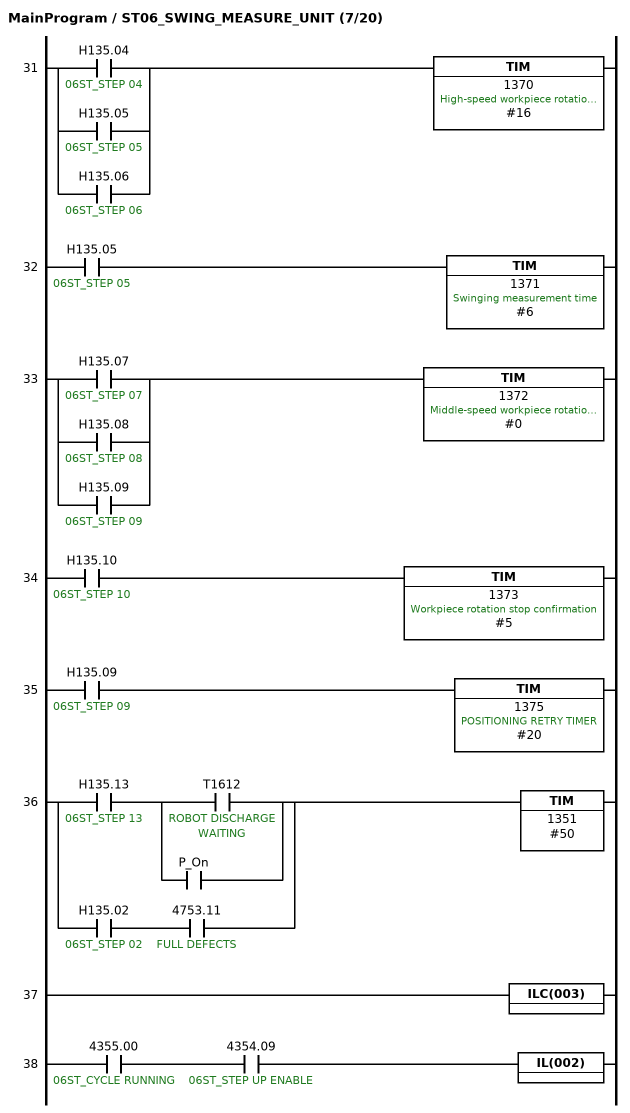
; [picture p360: MainProgram / ST06_SWING_MEASURE_UNIT, rungs 31-38]
; rung 31
LD H135.04  ; 06ST_STEP 04
OR H135.05  ; 06ST_STEP 05
OR H135.06  ; 06ST_STEP 06
TIM 1370 #16  ; High-speed workpiece rotation stability  // #15 => #8
; rung 32
LD H135.05  ; 06ST_STEP 05
TIM 1371 #6  ; Swinging measurement time
; rung 33
LD H135.07  ; 06ST_STEP 07
OR H135.08  ; 06ST_STEP 08
OR H135.09  ; 06ST_STEP 09
TIM 1372 #0  ; Middle-speed workpiece rotation stability
; rung 34
LD H135.10  ; 06ST_STEP 10
TIM 1373 #5  ; Workpiece rotation stop confirmation
; rung 35
LD H135.09  ; 06ST_STEP 09
TIM 1375 #20  ; POSITIONING RETRY TIMER
; rung 36
LD H135.13  ; 06ST_STEP 13
LD T1612  ; ROBOT DISCHARGE WAITING
OR P_On
ANDLD
LD H135.02  ; 06ST_STEP 02
AND 4753.11  ; FULL DEFECTS
ORLD
TIM 1351 #50
; rung 37
ILC(003)
; rung 38
LD 4355.00  ; 06ST_CYCLE RUNNING
AND 4354.09  ; 06ST_STEP UP ENABLE
IL(002)

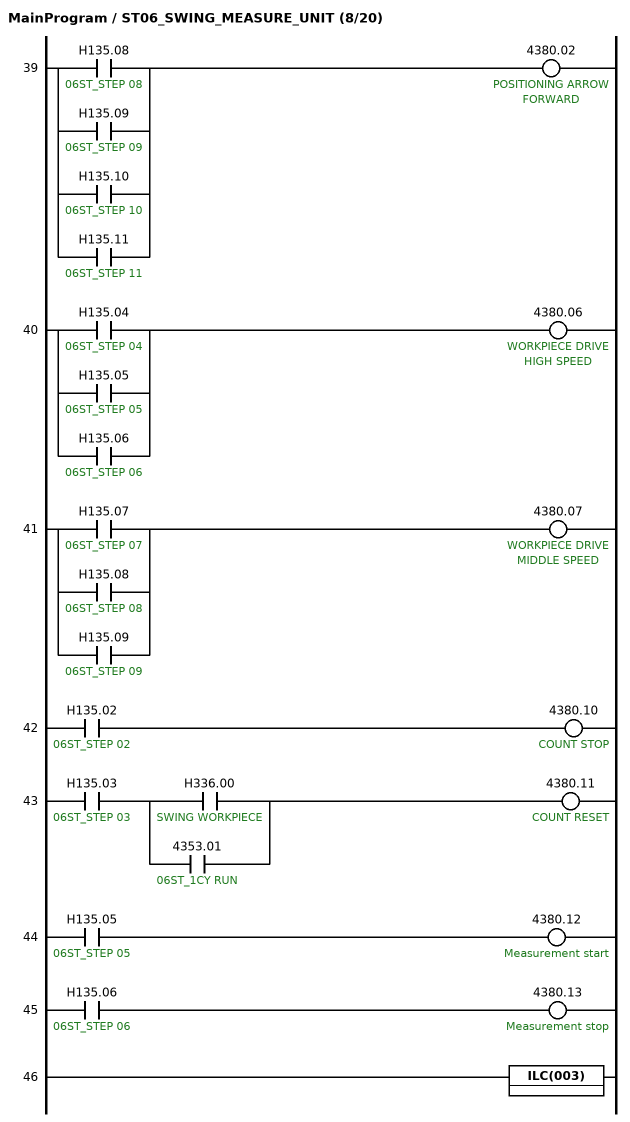
; rung 39
LD H135.08  ; 06ST_STEP 08
OR H135.09  ; 06ST_STEP 09
OR H135.10  ; 06ST_STEP 10
OR H135.11  ; 06ST_STEP 11
OUT 4380.02  ; POSITIONING ARROW FORWARD
; rung 40
LD H135.04  ; 06ST_STEP 04
OR H135.05  ; 06ST_STEP 05
OR H135.06  ; 06ST_STEP 06
OUT 4380.06  ; WORKPIECE DRIVE HIGH SPEED
; rung 41
LD H135.07  ; 06ST_STEP 07
OR H135.08  ; 06ST_STEP 08
OR H135.09  ; 06ST_STEP 09
OUT 4380.07  ; WORKPIECE DRIVE MIDDLE SPEED
; rung 42
LD H135.02  ; 06ST_STEP 02
OUT 4380.10  ; COUNT STOP
; rung 43
LD H135.03  ; 06ST_STEP 03
LD H336.00  ; SWING WORKPIECE
OR 4353.01  ; 06ST_1CY RUN
ANDLD
OUT 4380.11  ; COUNT RESET
; rung 44
LD H135.05  ; 06ST_STEP 05
OUT 4380.12  ; Measurement start
; rung 45
LD H135.06  ; 06ST_STEP 06
OUT 4380.13  ; Measurement stop
; rung 46
ILC(003)

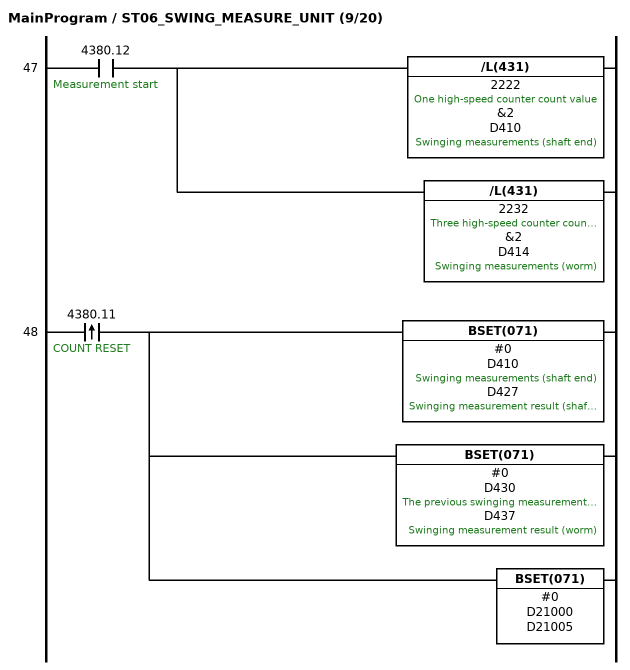
; rung 47
LD 4380.12  ; Measurement start
/L(431) 2222 &2 D410  ; One high-speed counter count value, Swinging measurements (shaft end)
/L(431) 2232 &2 D414  ; Three high-speed counter count value, Swinging measurements (worm)
; rung 48
@LD 4380.11  ; COUNT RESET
BSET(071) #0 D410 D427  ; Swinging measurements (shaft end), Swinging measurement result (shaft end)
BSET(071) #0 D430 D437  ; The previous swinging measurements (worm), Swinging measurement result (worm)
BSET(071) #0 D21000 D21005

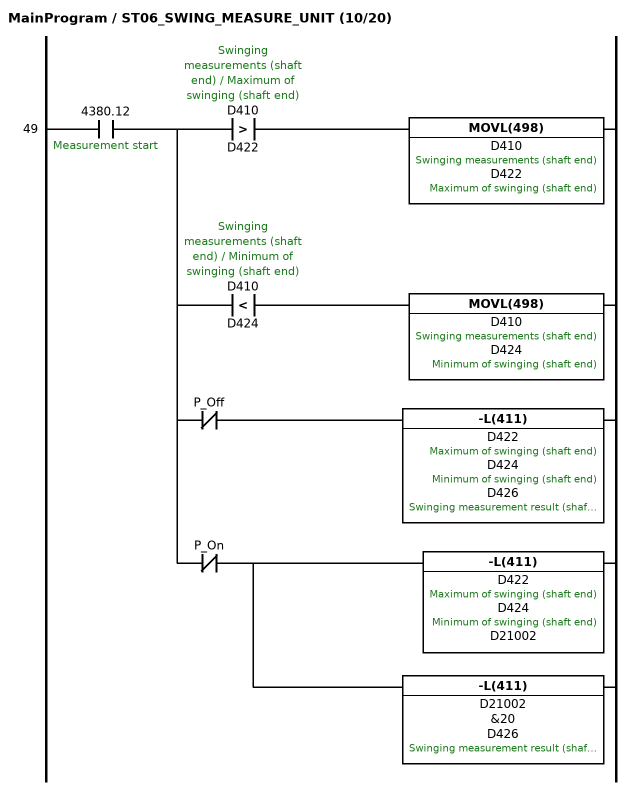
; rung 49
LD 4380.12  ; Measurement start
OUT TR0
AND>SL(323) D410 D422  ; Swinging measurements (shaft end), Maximum of swinging (shaft end)
MOVL(498) D410 D422  ; Swinging measurements (shaft end), Maximum of swinging (shaft end)
LD TR0
AND<SL(313) D410 D424  ; Swinging measurements (shaft end), Minimum of swinging (shaft end)
MOVL(498) D410 D424  ; Swinging measurements (shaft end), Minimum of swinging (shaft end)
LD TR0
ANDNOT P_Off
-L(411) D422 D424 D426  ; Maximum of swinging (shaft end), Minimum of swinging (shaft end), Swinging measurement result (shaft end)
LD TR0
ANDNOT P_On
-L(411) D422 D424 D21002  ; Maximum of swinging (shaft end), Minimum of swinging (shaft end)
-L(411) D21002 &20 D426  ; Swinging measurement result (shaft end)

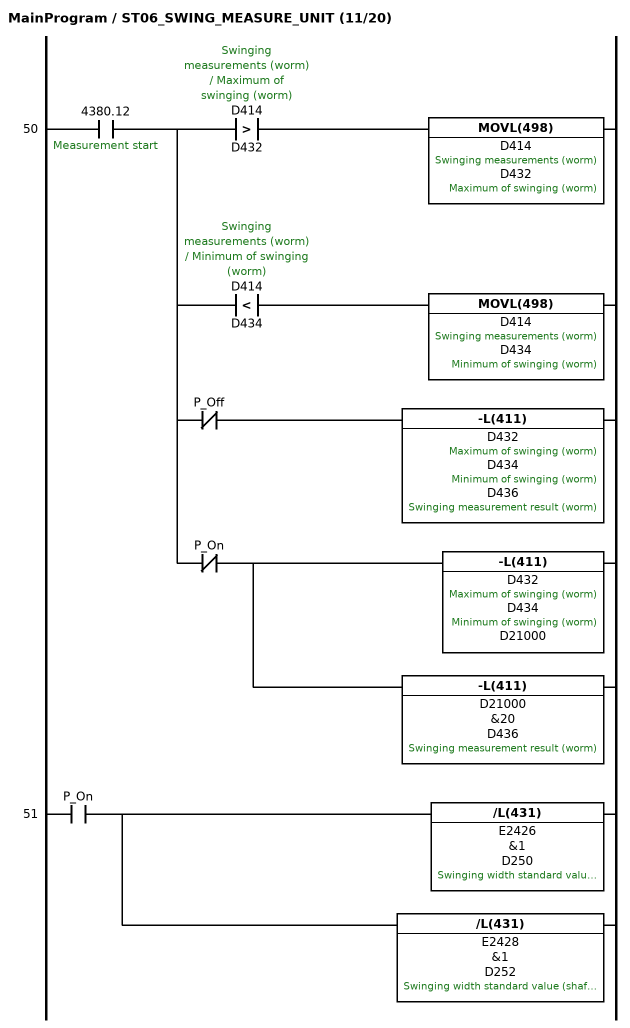
; rung 50
LD 4380.12  ; Measurement start
OUT TR0
AND>SL(323) D414 D432  ; Swinging measurements (worm), Maximum of swinging (worm)
MOVL(498) D414 D432  ; Swinging measurements (worm), Maximum of swinging (worm)
LD TR0
AND<SL(313) D414 D434  ; Swinging measurements (worm), Minimum of swinging (worm)
MOVL(498) D414 D434  ; Swinging measurements (worm), Minimum of swinging (worm)
LD TR0
ANDNOT P_Off
-L(411) D432 D434 D436  ; Maximum of swinging (worm), Minimum of swinging (worm), Swinging measurement result (worm)
LD TR0
ANDNOT P_On
-L(411) D432 D434 D21000  ; Maximum of swinging (worm), Minimum of swinging (worm)
-L(411) D21000 &20 D436  ; Swinging measurement result (worm)
; rung 51
LD P_On
/L(431) E2426 &1 D250  ; Swinging width standard value (worm)
/L(431) E2428 &1 D252  ; Swinging width standard value (shaft end)

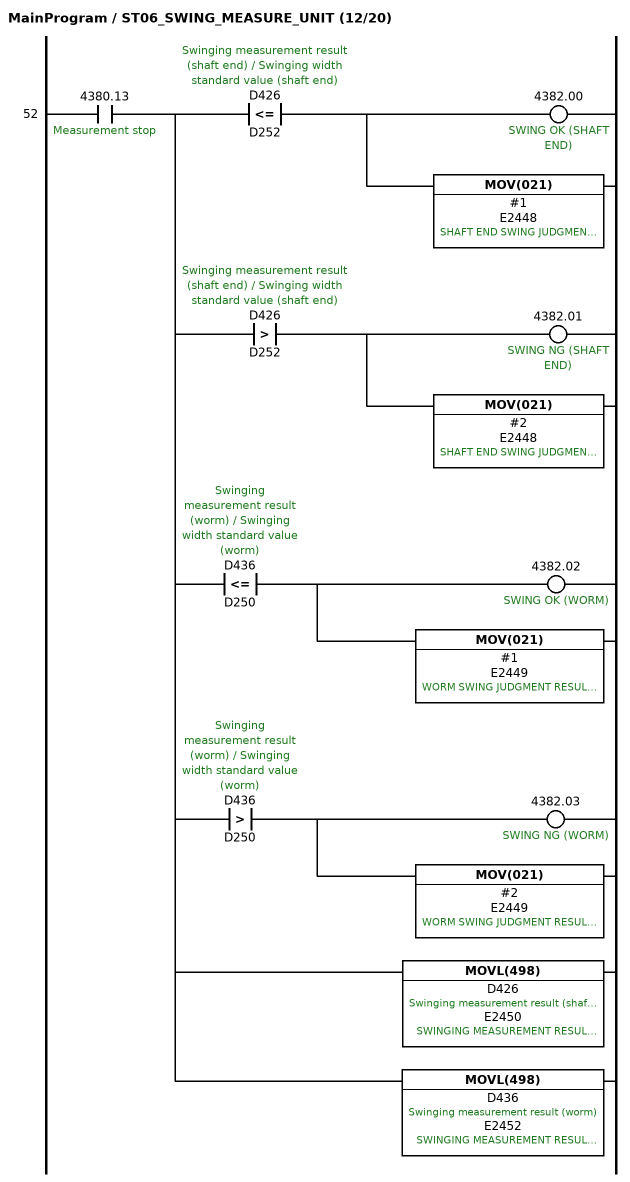
; rung 52
LD 4380.13  ; Measurement stop
OUT TR0
AND<=SL(318) D426 D252  ; Swinging measurement result (shaft end), Swinging width standard value (shaft end)
OUT 4382.00  ; SWING OK (SHAFT END)
MOV(021) #1 E2448  ; SHAFT END SWING JUDGMENT RESULT (1:OK,2:NG)
LD TR0
AND>SL(323) D426 D252  ; Swinging measurement result (shaft end), Swinging width standard value (shaft end)
OUT 4382.01  ; SWING NG (SHAFT END)
MOV(021) #2 E2448  ; SHAFT END SWING JUDGMENT RESULT (1:OK,2:NG)
LD TR0
AND<=SL(318) D436 D250  ; Swinging measurement result (worm), Swinging width standard value (worm)
OUT 4382.02  ; SWING OK (WORM)
MOV(021) #1 E2449  ; WORM SWING JUDGMENT RESULT (1:OK,2:NG)
LD TR0
AND>SL(323) D436 D250  ; Swinging measurement result (worm), Swinging width standard value (worm)
OUT 4382.03  ; SWING NG (WORM)
MOV(021) #2 E2449  ; WORM SWING JUDGMENT RESULT (1:OK,2:NG)
LD TR0
MOVL(498) D426 E2450  ; Swinging measurement result (shaft end), SWINGING MEASUREMENT RESULT (SHAFT END)
MOVL(498) D436 E2452  ; Swinging measurement result (worm), SWINGING MEASUREMENT RESULT (WORM)

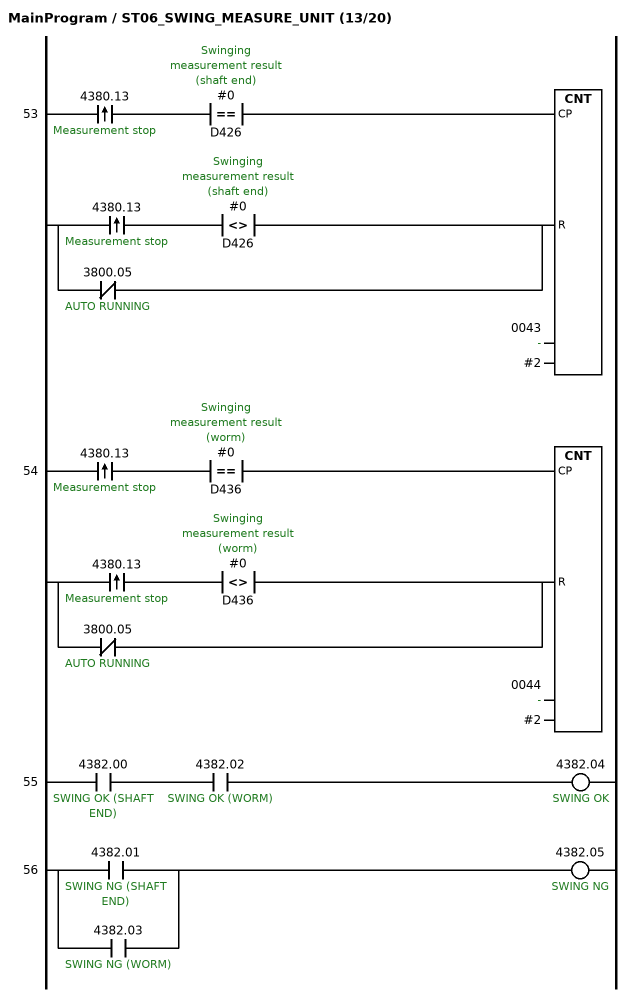
; rung 53
@LD 4380.13  ; Measurement stop
AND=SL(303) #0 D426  ; Swinging measurement result (shaft end)
@LD 4380.13  ; Measurement stop
AND<>SL(308) #0 D426  ; Swinging measurement result (shaft end)
ORNOT 3800.05  ; AUTO RUNNING
CNT 0043 #2  ; -
; rung 54
@LD 4380.13  ; Measurement stop
AND=SL(303) #0 D436  ; Swinging measurement result (worm)
@LD 4380.13  ; Measurement stop
AND<>SL(308) #0 D436  ; Swinging measurement result (worm)
ORNOT 3800.05  ; AUTO RUNNING
CNT 0044 #2  ; -
; rung 55
LD 4382.00  ; SWING OK (SHAFT END)
AND 4382.02  ; SWING OK (WORM)
OUT 4382.04  ; SWING OK
; rung 56
LD 4382.01  ; SWING NG (SHAFT END)
OR 4382.03  ; SWING NG (WORM)
OUT 4382.05  ; SWING NG

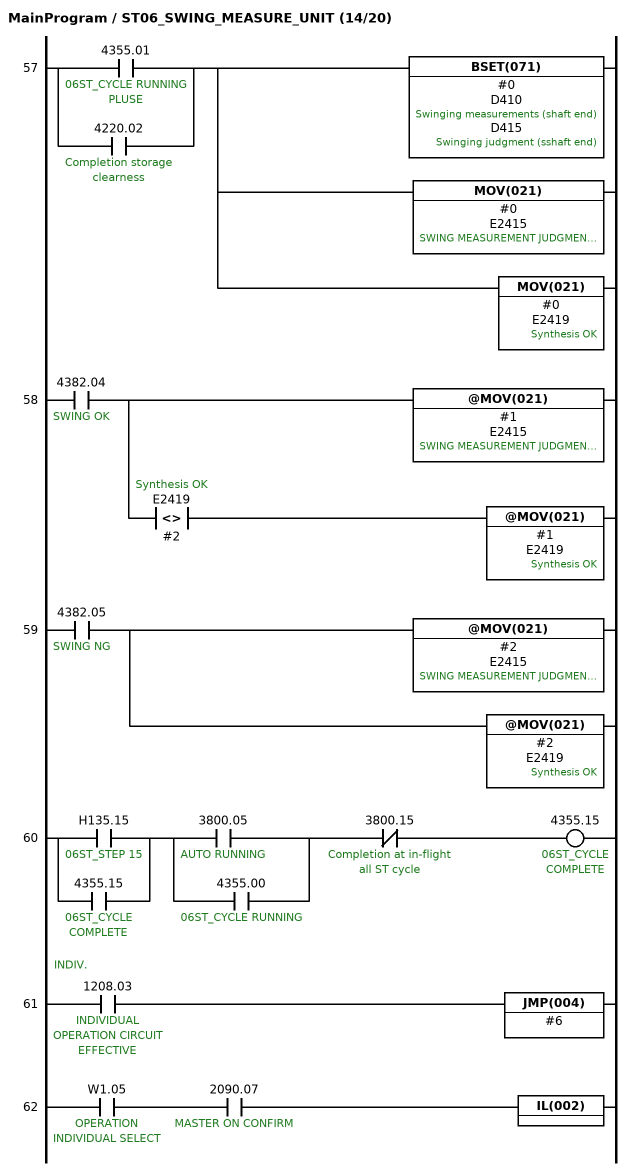
; rung 57
LD 4355.01  ; 06ST_CYCLE RUNNING PLUSE
OR 4220.02  ; Completion storage clearness
BSET(071) #0 D410 D415  ; Swinging measurements (shaft end), Swinging judgment (sshaft end)
MOV(021) #0 E2415  ; SWING MEASUREMENT JUDGMENT RESULT (1:OK,2:NG)
MOV(021) #0 E2419  ; Synthesis OK
; rung 58
LD 4382.04  ; SWING OK
@MOV(021) #1 E2415  ; SWING MEASUREMENT JUDGMENT RESULT (1:OK,2:NG)
AND<>(305) E2419 #2  ; Synthesis OK
@MOV(021) #1 E2419  ; Synthesis OK
; rung 59
LD 4382.05  ; SWING NG
@MOV(021) #2 E2415  ; SWING MEASUREMENT JUDGMENT RESULT (1:OK,2:NG)
@MOV(021) #2 E2419  ; Synthesis OK
; rung 60
LD H135.15  ; 06ST_STEP 15
OR 4355.15  ; 06ST_CYCLE COMPLETE
LD 3800.05  ; AUTO RUNNING
OR 4355.00  ; 06ST_CYCLE RUNNING
ANDLD
ANDNOT 3800.15  ; Completion at in-flight all ST cycle
OUT 4355.15  ; 06ST_CYCLE COMPLETE
; rung 61: INDIV.
LD 1208.03  ; INDIVIDUAL OPERATION CIRCUIT EFFECTIVE
JMP(004) #6
; rung 62
LD W1.05  ; OPERATION INDIVIDUAL SELECT
AND 2090.07  ; MASTER ON CONFIRM
IL(002)

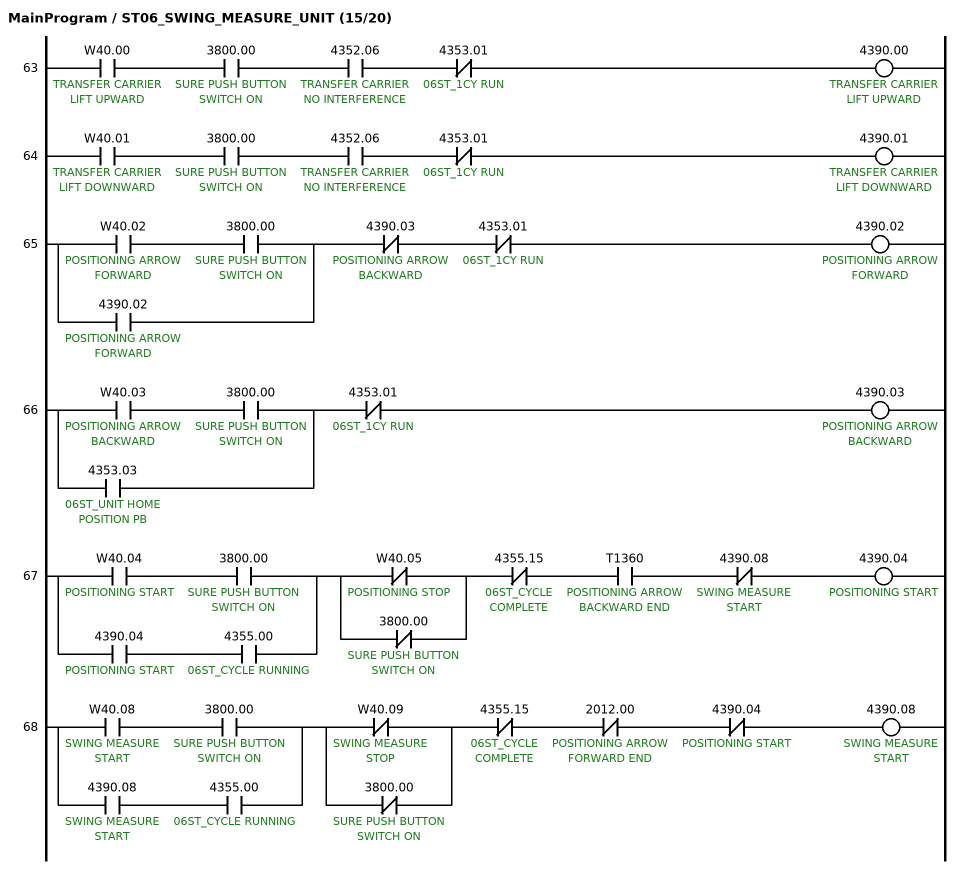
; rung 63
LD W40.00  ; TRANSFER CARRIER LIFT UPWARD
AND 3800.00  ; SURE PUSH BUTTON SWITCH ON
AND 4352.06  ; TRANSFER CARRIER NO INTERFERENCE
ANDNOT 4353.01  ; 06ST_1CY RUN
OUT 4390.00  ; TRANSFER CARRIER LIFT UPWARD
; rung 64
LD W40.01  ; TRANSFER CARRIER LIFT DOWNWARD
AND 3800.00  ; SURE PUSH BUTTON SWITCH ON
AND 4352.06  ; TRANSFER CARRIER NO INTERFERENCE
ANDNOT 4353.01  ; 06ST_1CY RUN
OUT 4390.01  ; TRANSFER CARRIER LIFT DOWNWARD
; rung 65
LD W40.02  ; POSITIONING ARROW FORWARD
AND 3800.00  ; SURE PUSH BUTTON SWITCH ON
OR 4390.02  ; POSITIONING ARROW FORWARD
ANDNOT 4390.03  ; POSITIONING ARROW BACKWARD
ANDNOT 4353.01  ; 06ST_1CY RUN
OUT 4390.02  ; POSITIONING ARROW FORWARD
; rung 66
LD W40.03  ; POSITIONING ARROW BACKWARD
AND 3800.00  ; SURE PUSH BUTTON SWITCH ON
OR 4353.03  ; 06ST_UNIT HOME POSITION PB
ANDNOT 4353.01  ; 06ST_1CY RUN
OUT 4390.03  ; POSITIONING ARROW BACKWARD
; rung 67
LD W40.04  ; POSITIONING START
AND 3800.00  ; SURE PUSH BUTTON SWITCH ON
LD 4390.04  ; POSITIONING START
AND 4355.00  ; 06ST_CYCLE RUNNING
ORLD
LDNOT W40.05  ; POSITIONING STOP
ORNOT 3800.00  ; SURE PUSH BUTTON SWITCH ON
ANDLD
ANDNOT 4355.15  ; 06ST_CYCLE COMPLETE
AND T1360  ; POSITIONING ARROW BACKWARD END
ANDNOT 4390.08  ; SWING MEASURE START
OUT 4390.04  ; POSITIONING START
; rung 68
LD W40.08  ; SWING MEASURE START
AND 3800.00  ; SURE PUSH BUTTON SWITCH ON
LD 4390.08  ; SWING MEASURE START
AND 4355.00  ; 06ST_CYCLE RUNNING
ORLD
LDNOT W40.09  ; SWING MEASURE STOP
ORNOT 3800.00  ; SURE PUSH BUTTON SWITCH ON
ANDLD
ANDNOT 4355.15  ; 06ST_CYCLE COMPLETE
ANDNOT 2012.00  ; POSITIONING ARROW FORWARD END
ANDNOT 4390.04  ; POSITIONING START
OUT 4390.08  ; SWING MEASURE START

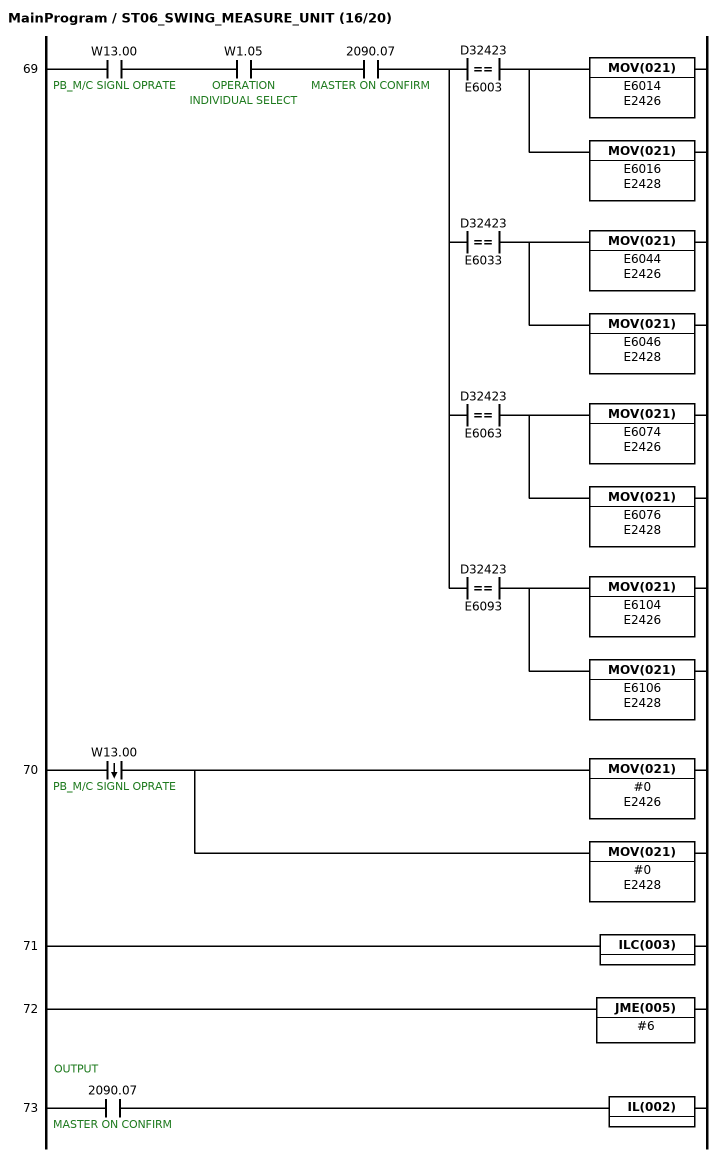
; rung 69
LD W13.00  ; PB_M/C SIGNL OPRATE
AND W1.05  ; OPERATION INDIVIDUAL SELECT
AND 2090.07  ; MASTER ON CONFIRM
OUT TR0
AND=(300) D32423 E6003
MOV(021) E6014 E2426
MOV(021) E6016 E2428
LD TR0
AND=(300) D32423 E6033
MOV(021) E6044 E2426
MOV(021) E6046 E2428
LD TR0
AND=(300) D32423 E6063
MOV(021) E6074 E2426
MOV(021) E6076 E2428
LD TR0
AND=(300) D32423 E6093
MOV(021) E6104 E2426
MOV(021) E6106 E2428
; rung 70
%LD W13.00  ; PB_M/C SIGNL OPRATE
MOV(021) #0 E2426
MOV(021) #0 E2428
; rung 71
ILC(003)
; rung 72
JME(005) #6
; rung 73: OUTPUT
LD 2090.07  ; MASTER ON CONFIRM
IL(002)

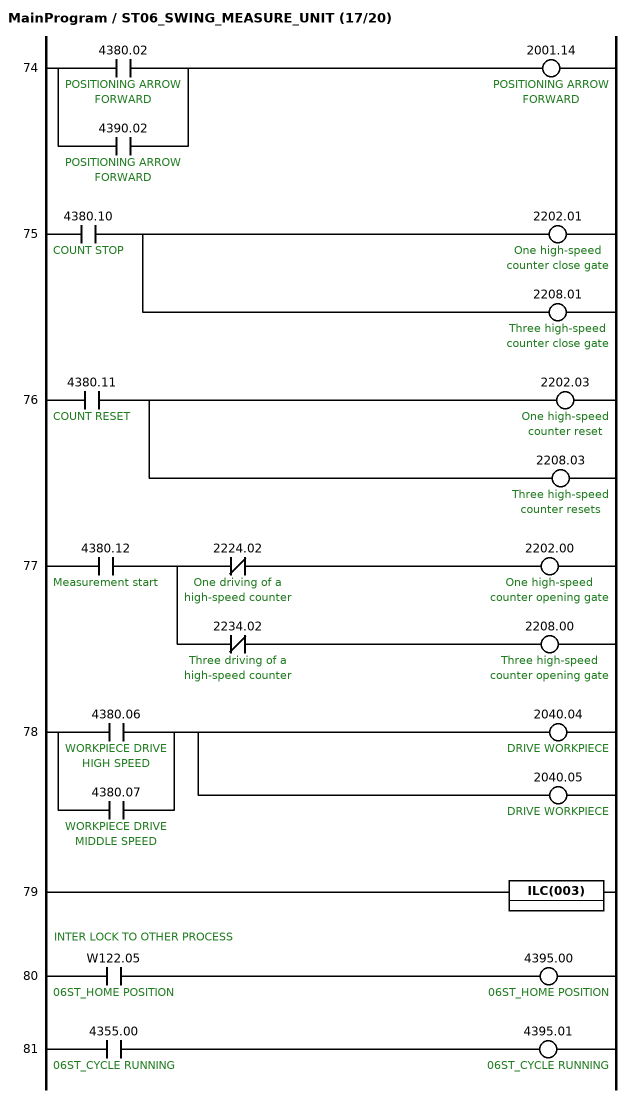
; rung 74
LD 4380.02  ; POSITIONING ARROW FORWARD
OR 4390.02  ; POSITIONING ARROW FORWARD
OUT 2001.14  ; POSITIONING ARROW FORWARD
; rung 75
LD 4380.10  ; COUNT STOP
OUT 2202.01  ; One high-speed counter close gate
OUT 2208.01  ; Three high-speed counter close gate
; rung 76
LD 4380.11  ; COUNT RESET
OUT 2202.03  ; One high-speed counter reset
OUT 2208.03  ; Three high-speed counter resets
; rung 77
LD 4380.12  ; Measurement start
OUT TR0
ANDNOT 2224.02  ; One driving of a high-speed counter
OUT 2202.00  ; One high-speed counter opening gate
LD TR0
ANDNOT 2234.02  ; Three driving of a high-speed counter
OUT 2208.00  ; Three high-speed counter opening gate
; rung 78
LD 4380.06  ; WORKPIECE DRIVE HIGH SPEED
OR 4380.07  ; WORKPIECE DRIVE MIDDLE SPEED
OUT 2040.04  ; DRIVE WORKPIECE
OUT 2040.05  ; DRIVE WORKPIECE
; rung 79
ILC(003)
; rung 80: INTER LOCK TO OTHER PROCESS
LD W122.05  ; 06ST_HOME POSITION
OUT 4395.00  ; 06ST_HOME POSITION
; rung 81
LD 4355.00  ; 06ST_CYCLE RUNNING
OUT 4395.01  ; 06ST_CYCLE RUNNING

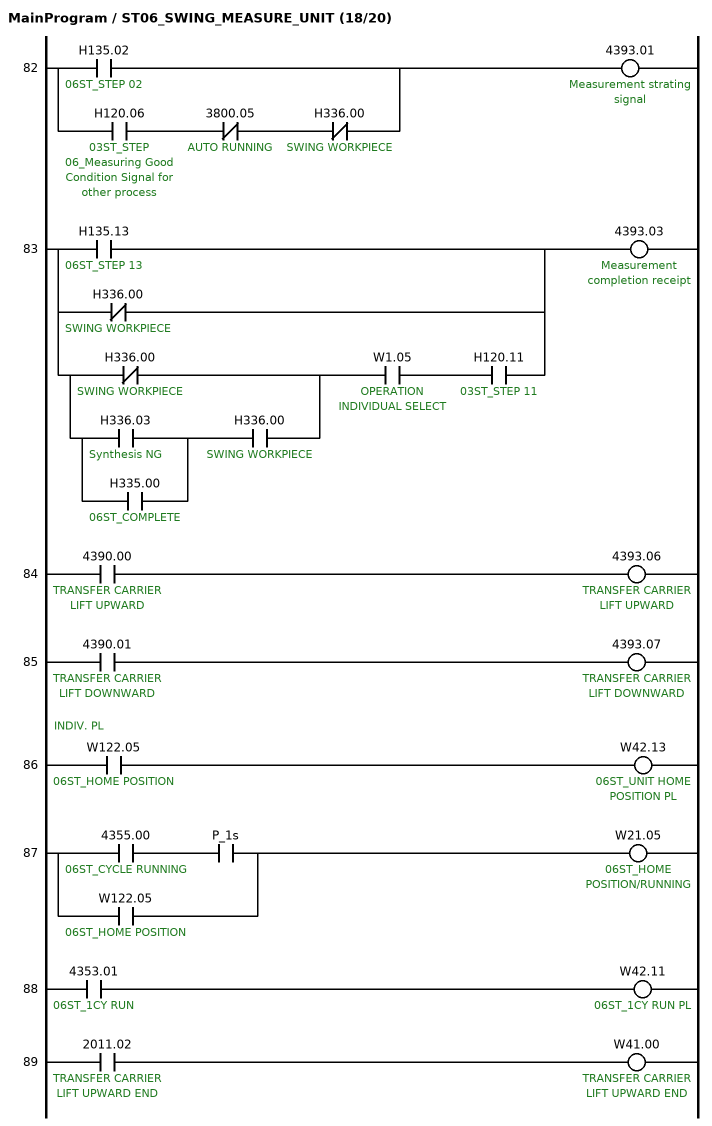
; rung 82
LD H135.02  ; 06ST_STEP 02
LD H120.06  ; 03ST_STEP 06_Measuring Good Condition Signal for other process
ANDNOT 3800.05  ; AUTO RUNNING
ANDNOT H336.00  ; SWING WORKPIECE
ORLD
OUT 4393.01  ; Measurement strating signal
; rung 83
LD H135.13  ; 06ST_STEP 13
ORNOT H336.00  ; SWING WORKPIECE
LDNOT H336.00  ; SWING WORKPIECE
LD H336.03  ; Synthesis NG
OR H335.00  ; 06ST_COMPLETE
AND H336.00  ; SWING WORKPIECE
ORLD
AND W1.05  ; OPERATION INDIVIDUAL SELECT
AND H120.11  ; 03ST_STEP 11
ORLD
OUT 4393.03  ; Measurement completion receipt
; rung 84
LD 4390.00  ; TRANSFER CARRIER LIFT UPWARD
OUT 4393.06  ; TRANSFER CARRIER LIFT UPWARD
; rung 85
LD 4390.01  ; TRANSFER CARRIER LIFT DOWNWARD
OUT 4393.07  ; TRANSFER CARRIER LIFT DOWNWARD
; rung 86: INDIV. PL
LD W122.05  ; 06ST_HOME POSITION
OUT W42.13  ; 06ST_UNIT HOME POSITION PL
; rung 87
LD 4355.00  ; 06ST_CYCLE RUNNING
AND P_1s
OR W122.05  ; 06ST_HOME POSITION
OUT W21.05  ; 06ST_HOME POSITION/RUNNING
; rung 88
LD 4353.01  ; 06ST_1CY RUN
OUT W42.11  ; 06ST_1CY RUN PL
; rung 89
LD 2011.02  ; TRANSFER CARRIER LIFT UPWARD END
OUT W41.00  ; TRANSFER CARRIER LIFT UPWARD END

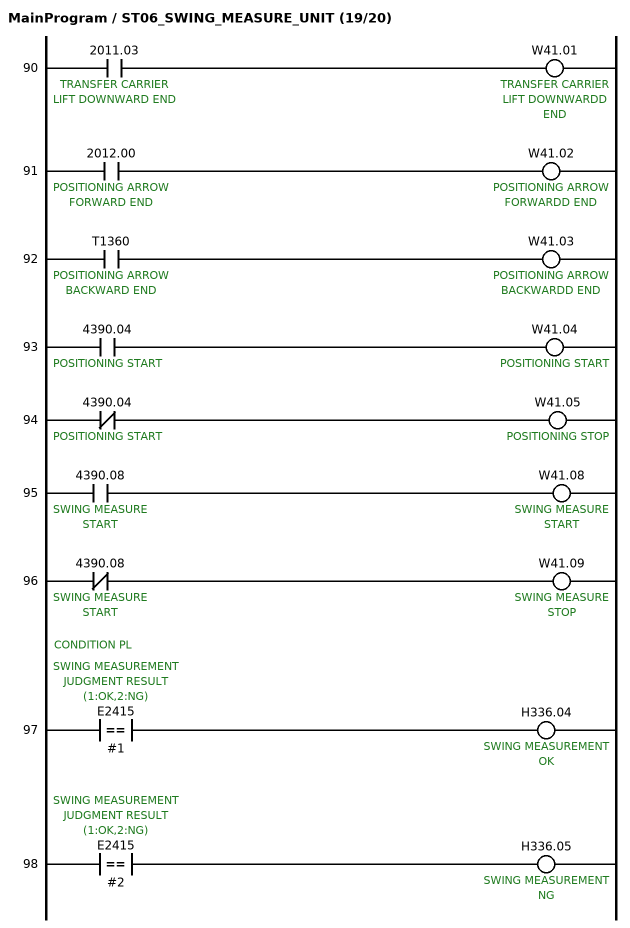
; rung 90
LD 2011.03  ; TRANSFER CARRIER LIFT DOWNWARD END
OUT W41.01  ; TRANSFER CARRIER LIFT DOWNWARDD END
; rung 91
LD 2012.00  ; POSITIONING ARROW FORWARD END
OUT W41.02  ; POSITIONING ARROW FORWARDD END
; rung 92
LD T1360  ; POSITIONING ARROW BACKWARD END
OUT W41.03  ; POSITIONING ARROW BACKWARDD END
; rung 93
LD 4390.04  ; POSITIONING START
OUT W41.04  ; POSITIONING START
; rung 94
LDNOT 4390.04  ; POSITIONING START
OUT W41.05  ; POSITIONING STOP
; rung 95
LD 4390.08  ; SWING MEASURE START
OUT W41.08  ; SWING MEASURE START
; rung 96
LDNOT 4390.08  ; SWING MEASURE START
OUT W41.09  ; SWING MEASURE STOP
; rung 97: CONDITION PL
LD=(300) E2415 #1  ; SWING MEASUREMENT JUDGMENT RESULT (1:OK,2:NG)
OUT H336.04  ; SWING MEASUREMENT OK
; rung 98
LD=(300) E2415 #2  ; SWING MEASUREMENT JUDGMENT RESULT (1:OK,2:NG)
OUT H336.05  ; SWING MEASUREMENT NG

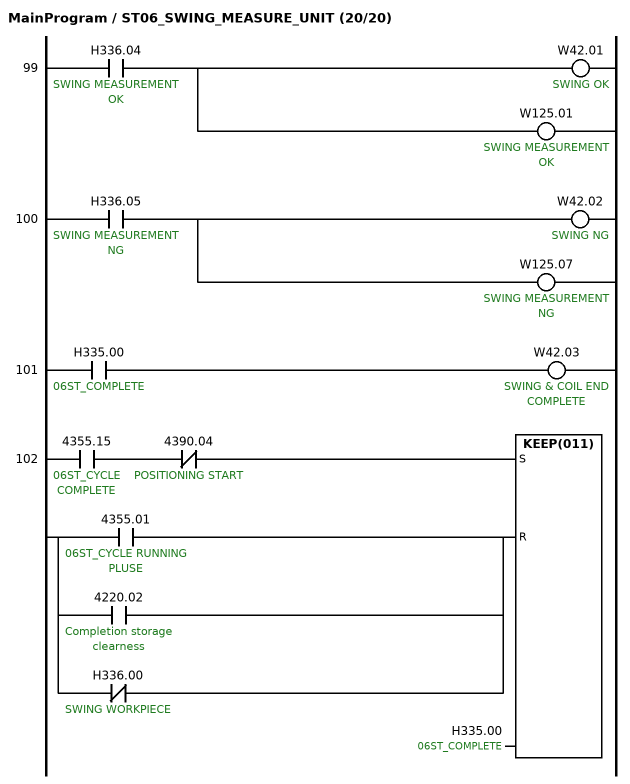
; rung 99
LD H336.04  ; SWING MEASUREMENT OK
OUT W42.01  ; SWING OK
OUT W125.01  ; SWING MEASUREMENT OK
; rung 100
LD H336.05  ; SWING MEASUREMENT NG
OUT W42.02  ; SWING NG
OUT W125.07  ; SWING MEASUREMENT NG
; rung 101
LD H335.00  ; 06ST_COMPLETE
OUT W42.03  ; SWING & COIL END COMPLETE
; rung 102
LD 4355.15  ; 06ST_CYCLE COMPLETE
ANDNOT 4390.04  ; POSITIONING START
LD 4355.01  ; 06ST_CYCLE RUNNING PLUSE
OR 4220.02  ; Completion storage clearness
ORNOT H336.00  ; SWING WORKPIECE
KEEP(011) H335.00  ; 06ST_COMPLETE

### Section ST07_RESISTANSE_UNIT

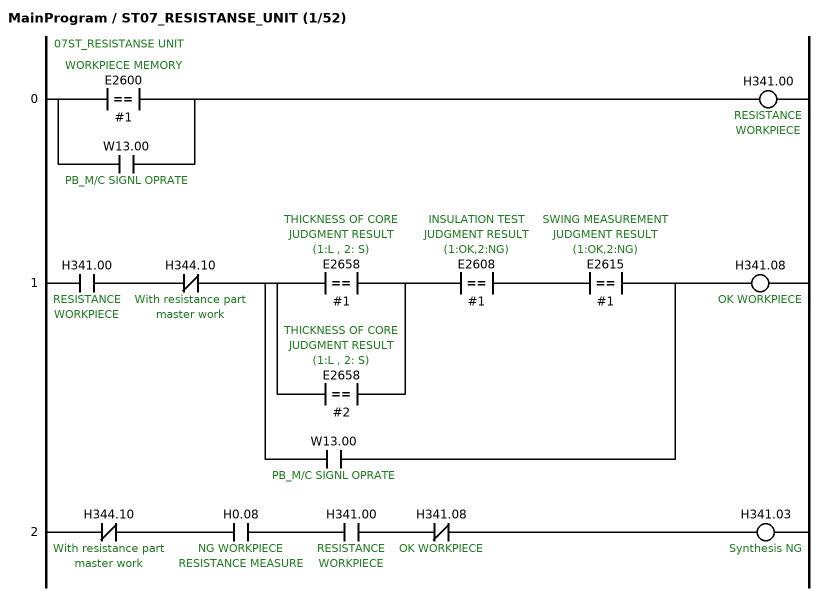
; rung 0: 07ST_RESISTANSE UNIT
LD=(300) E2600 #1  ; WORKPIECE MEMORY
OR W13.00  ; PB_M/C SIGNL OPRATE
OUT H341.00  ; RESISTANCE WORKPIECE
; rung 1
LD H341.00  ; RESISTANCE WORKPIECE
ANDNOT H344.10  ; With resistance part master work
LD=(300) E2658 #1  ; THICKNESS OF CORE JUDGMENT RESULT (1:L , 2: S)
OR=(300) E2658 #2  ; THICKNESS OF CORE JUDGMENT RESULT (1:L , 2: S)
AND=(300) E2608 #1  ; INSULATION TEST JUDGMENT RESULT (1:OK,2:NG)
AND=(300) E2615 #1  ; SWING MEASUREMENT JUDGMENT RESULT (1:OK,2:NG)
OR W13.00  ; PB_M/C SIGNL OPRATE
ANDLD
OUT H341.08  ; OK WORKPIECE
; rung 2
LDNOT H344.10  ; With resistance part master work
AND H0.08  ; NG WORKPIECE RESISTANCE MEASURE
AND H341.00  ; RESISTANCE WORKPIECE
ANDNOT H341.08  ; OK WORKPIECE
OUT H341.03  ; Synthesis NG

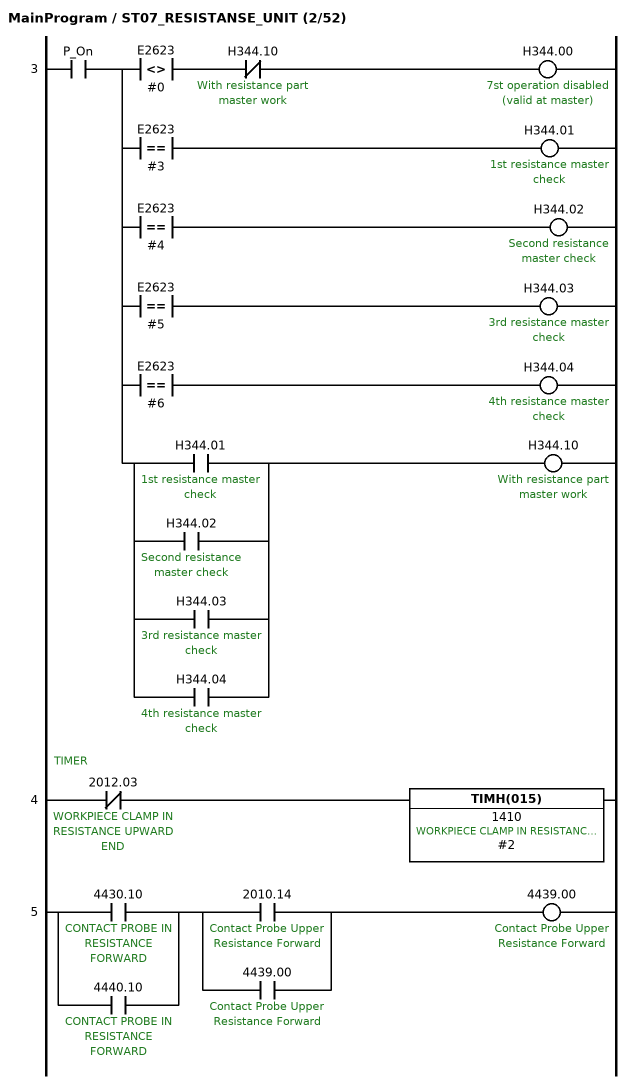
; rung 3
LD P_On
OUT TR0
AND<>(305) E2623 #0
ANDNOT H344.10  ; With resistance part master work
OUT H344.00  ; 7st operation disabled (valid at master)
LD TR0
AND=(300) E2623 #3
OUT H344.01  ; 1st resistance master check
LD TR0
AND=(300) E2623 #4
OUT H344.02  ; Second resistance master check
LD TR0
AND=(300) E2623 #5
OUT H344.03  ; 3rd resistance master check
LD TR0
AND=(300) E2623 #6
OUT H344.04  ; 4th resistance master check
LD TR0
LD H344.01  ; 1st resistance master check
OR H344.02  ; Second resistance master check
OR H344.03  ; 3rd resistance master check
OR H344.04  ; 4th resistance master check
ANDLD
OUT H344.10  ; With resistance part master work
; rung 4: TIMER
LDNOT 2012.03  ; WORKPIECE CLAMP IN RESISTANCE UPWARD END
TIMH(015) 1410 #2  ; WORKPIECE CLAMP IN RESISTANCE DOWNWARD END
; rung 5
LD 4430.10  ; CONTACT PROBE IN RESISTANCE FORWARD
OR 4440.10  ; CONTACT PROBE IN RESISTANCE FORWARD
LD 2010.14  ; Contact Probe Upper Resistance Forward
OR 4439.00  ; Contact Probe Upper Resistance Forward
ANDLD
OUT 4439.00  ; Contact Probe Upper Resistance Forward

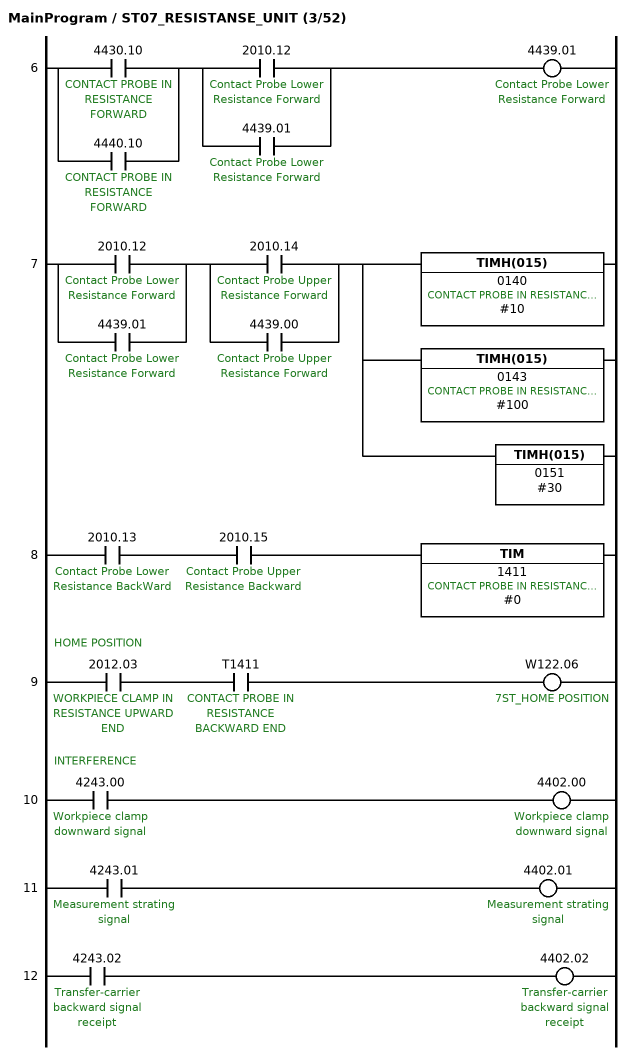
; rung 6
LD 4430.10  ; CONTACT PROBE IN RESISTANCE FORWARD
OR 4440.10  ; CONTACT PROBE IN RESISTANCE FORWARD
LD 2010.12  ; Contact Probe Lower Resistance Forward
OR 4439.01  ; Contact Probe Lower Resistance Forward
ANDLD
OUT 4439.01  ; Contact Probe Lower Resistance Forward
; rung 7
LD 2010.12  ; Contact Probe Lower Resistance Forward
OR 4439.01  ; Contact Probe Lower Resistance Forward
LD 2010.14  ; Contact Probe Upper Resistance Forward
OR 4439.00  ; Contact Probe Upper Resistance Forward
ANDLD
TIMH(015) 0140 #10  ; CONTACT PROBE IN RESISTANCE FORWARD END
TIMH(015) 0143 #100  ; CONTACT PROBE IN RESISTANCE FORWARD END
TIMH(015) 0151 #30
; rung 8
LD 2010.13  ; Contact Probe Lower Resistance BackWard
AND 2010.15  ; Contact Probe Upper Resistance Backward
TIM 1411 #0  ; CONTACT PROBE IN RESISTANCE BACKWARD END  // #2 => #0
; rung 9: HOME POSITION
LD 2012.03  ; WORKPIECE CLAMP IN RESISTANCE UPWARD END
AND T1411  ; CONTACT PROBE IN RESISTANCE BACKWARD END
OUT W122.06  ; 7ST_HOME POSITION
; rung 10: INTERFERENCE
LD 4243.00  ; Workpiece clamp downward signal
OUT 4402.00  ; Workpiece clamp downward signal
; rung 11
LD 4243.01  ; Measurement strating signal
OUT 4402.01  ; Measurement strating signal
; rung 12
LD 4243.02  ; Transfer-carrier backward signal receipt
OUT 4402.02  ; Transfer-carrier backward signal receipt

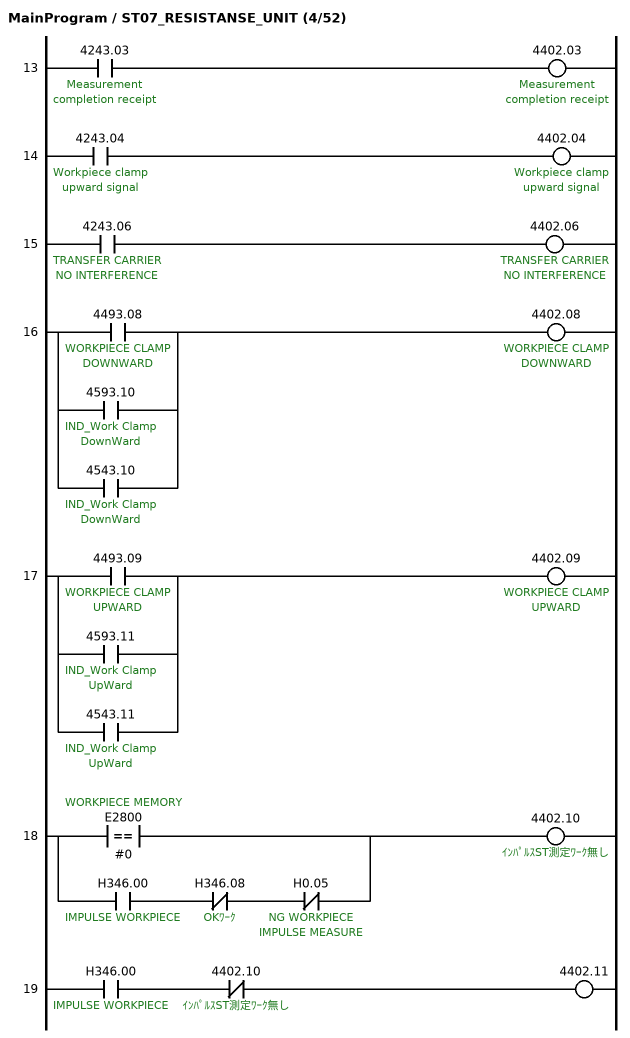
; rung 13
LD 4243.03  ; Measurement completion receipt
OUT 4402.03  ; Measurement completion receipt
; rung 14
LD 4243.04  ; Workpiece clamp upward signal
OUT 4402.04  ; Workpiece clamp upward signal
; rung 15
LD 4243.06  ; TRANSFER CARRIER NO INTERFERENCE
OUT 4402.06  ; TRANSFER CARRIER NO INTERFERENCE
; rung 16
LD 4493.08  ; WORKPIECE CLAMP DOWNWARD
OR 4593.10  ; IND_Work Clamp DownWard
OR 4543.10  ; IND_Work Clamp DownWard
OUT 4402.08  ; WORKPIECE CLAMP DOWNWARD
; rung 17
LD 4493.09  ; WORKPIECE CLAMP UPWARD
OR 4593.11  ; IND_Work Clamp UpWard
OR 4543.11  ; IND_Work Clamp UpWard
OUT 4402.09  ; WORKPIECE CLAMP UPWARD
; rung 18
LD=(300) E2800 #0  ; WORKPIECE MEMORY
LD H346.00  ; IMPULSE WORKPIECE
ANDNOT H346.08  ; OKﾜｰｸ
ANDNOT H0.05  ; NG WORKPIECE IMPULSE MEASURE
ORLD
OUT 4402.10  ; ｲﾝﾊﾟﾙｽST測定ﾜｰｸ無し
; rung 19
LD H346.00  ; IMPULSE WORKPIECE
ANDNOT 4402.10  ; ｲﾝﾊﾟﾙｽST測定ﾜｰｸ無し
OUT 4402.11

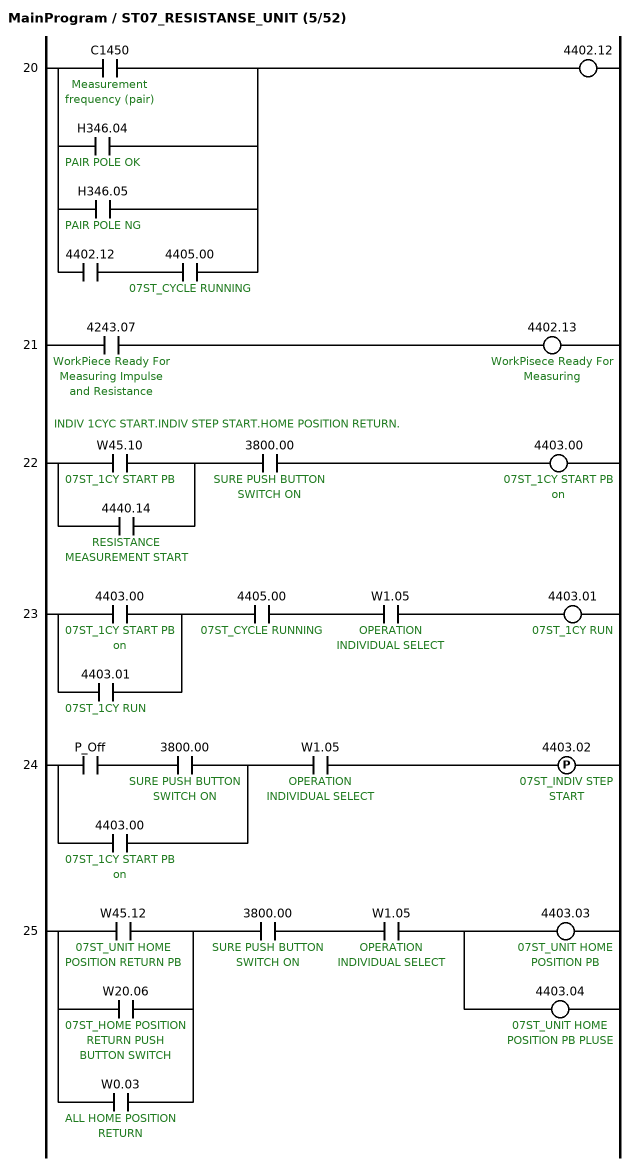
; rung 20
LD C1450  ; Measurement frequency (pair)
OR H346.04  ; PAIR POLE OK
OR H346.05  ; PAIR POLE NG
LD 4402.12
AND 4405.00  ; 07ST_CYCLE RUNNING
ORLD
OUT 4402.12
; rung 21
LD 4243.07  ; WorkPiece Ready For Measuring Impulse and Resistance
OUT 4402.13  ; WorkPisece Ready For Measuring
; rung 22: INDIV 1CYC START.INDIV STEP START.HOME POSITION RETURN.
LD W45.10  ; 07ST_1CY START PB
OR 4440.14  ; RESISTANCE MEASUREMENT START
AND 3800.00  ; SURE PUSH BUTTON SWITCH ON
OUT 4403.00  ; 07ST_1CY START PB on
; rung 23
LD 4403.00  ; 07ST_1CY START PB on
OR 4403.01  ; 07ST_1CY RUN
AND 4405.00  ; 07ST_CYCLE RUNNING
AND W1.05  ; OPERATION INDIVIDUAL SELECT
OUT 4403.01  ; 07ST_1CY RUN
; rung 24
LD P_Off
AND 3800.00  ; SURE PUSH BUTTON SWITCH ON
OR 4403.00  ; 07ST_1CY START PB on
AND W1.05  ; OPERATION INDIVIDUAL SELECT
DIFU(013) 4403.02  ; 07ST_INDIV STEP START
; rung 25
LD W45.12  ; 07ST_UNIT HOME POSITION RETURN PB
OR W20.06  ; 07ST_HOME POSITION RETURN PUSH BUTTON SWITCH
OR W0.03  ; ALL HOME POSITION RETURN
AND 3800.00  ; SURE PUSH BUTTON SWITCH ON
AND W1.05  ; OPERATION INDIVIDUAL SELECT
OUT 4403.03  ; 07ST_UNIT HOME POSITION PB
OUT 4403.04  ; 07ST_UNIT HOME POSITION PB PLUSE

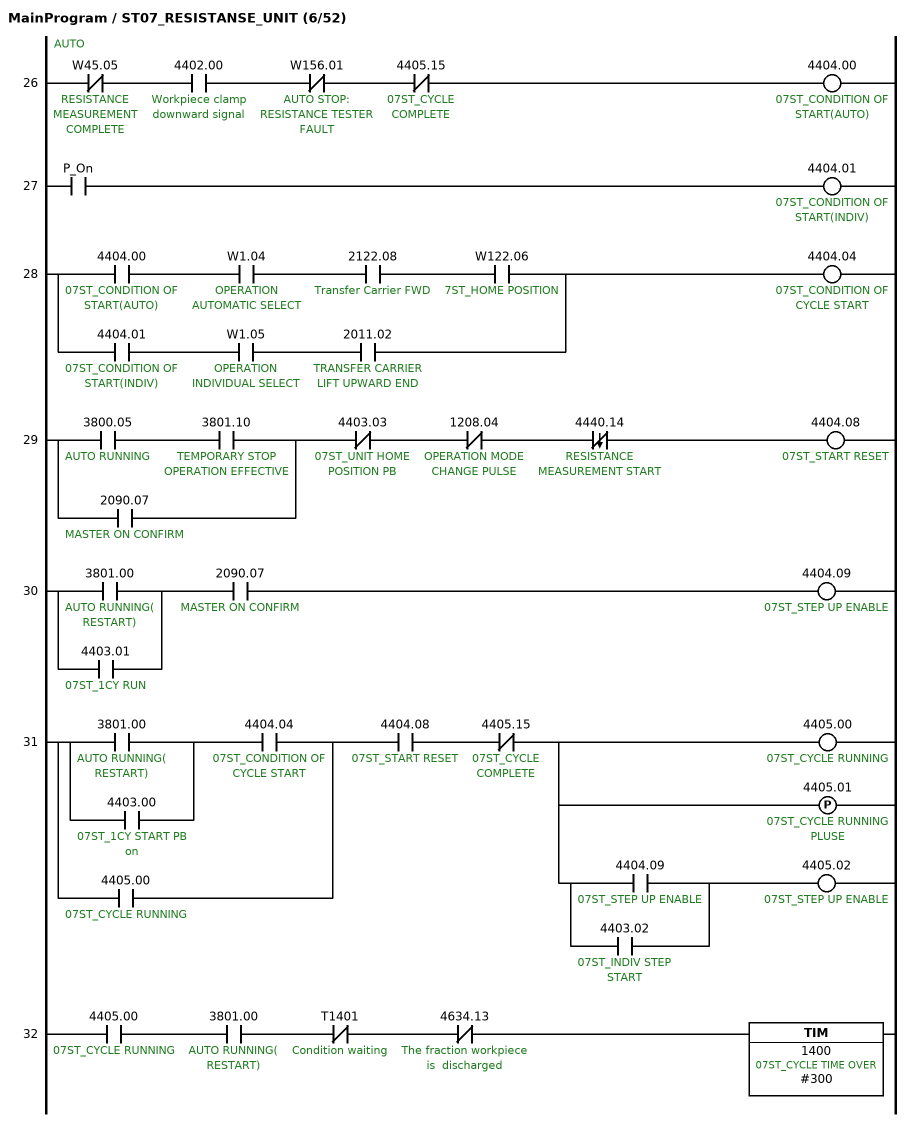
; rung 26: AUTO
LDNOT W45.05  ; RESISTANCE MEASUREMENT COMPLETE
AND 4402.00  ; Workpiece clamp downward signal
ANDNOT W156.01  ; AUTO STOP:RESISTANCE TESTER FAULT
ANDNOT 4405.15  ; 07ST_CYCLE COMPLETE
OUT 4404.00  ; 07ST_CONDITION OF START(AUTO)
; rung 27
LD P_On
OUT 4404.01  ; 07ST_CONDITION OF START(INDIV)
; rung 28
LD 4404.00  ; 07ST_CONDITION OF START(AUTO)
AND W1.04  ; OPERATION AUTOMATIC SELECT
AND 2122.08  ; Transfer Carrier FWD
AND W122.06  ; 7ST_HOME POSITION
LD 4404.01  ; 07ST_CONDITION OF START(INDIV)
AND W1.05  ; OPERATION INDIVIDUAL SELECT
AND 2011.02  ; TRANSFER CARRIER LIFT UPWARD END
ORLD
OUT 4404.04  ; 07ST_CONDITION OF CYCLE START
; rung 29
LD 3800.05  ; AUTO RUNNING
AND 3801.10  ; TEMPORARY STOP OPERATION EFFECTIVE
OR 2090.07  ; MASTER ON CONFIRM
ANDNOT 4403.03  ; 07ST_UNIT HOME POSITION PB
ANDNOT 1208.04  ; OPERATION MODE CHANGE PULSE
%ANDNOT 4440.14  ; RESISTANCE MEASUREMENT START
OUT 4404.08  ; 07ST_START RESET
; rung 30
LD 3801.00  ; AUTO RUNNING(RESTART)
OR 4403.01  ; 07ST_1CY RUN
AND 2090.07  ; MASTER ON CONFIRM
OUT 4404.09  ; 07ST_STEP UP ENABLE
; rung 31
LD 3801.00  ; AUTO RUNNING(RESTART)
OR 4403.00  ; 07ST_1CY START PB on
AND 4404.04  ; 07ST_CONDITION OF CYCLE START
OR 4405.00  ; 07ST_CYCLE RUNNING
AND 4404.08  ; 07ST_START RESET
ANDNOT 4405.15  ; 07ST_CYCLE COMPLETE
OUT 4405.00  ; 07ST_CYCLE RUNNING
DIFU(013) 4405.01  ; 07ST_CYCLE RUNNING PLUSE
LD 4404.09  ; 07ST_STEP UP ENABLE
OR 4403.02  ; 07ST_INDIV STEP START
ANDLD
OUT 4405.02  ; 07ST_STEP UP ENABLE
; rung 32
LD 4405.00  ; 07ST_CYCLE RUNNING
AND 3801.00  ; AUTO RUNNING(RESTART)
ANDNOT T1401  ; Condition waiting
ANDNOT 4634.13  ; The fraction workpiece is  discharged
TIM 1400 #300  ; 07ST_CYCLE TIME OVER

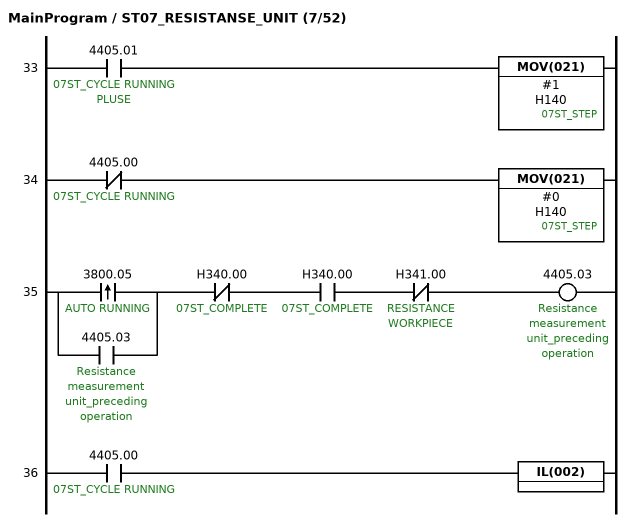
; rung 33
LD 4405.01  ; 07ST_CYCLE RUNNING PLUSE
MOV(021) #1 H140  ; 07ST_STEP
; rung 34
LDNOT 4405.00  ; 07ST_CYCLE RUNNING
MOV(021) #0 H140  ; 07ST_STEP
; rung 35
@LD 3800.05  ; AUTO RUNNING
OR 4405.03  ; Resistance measurement unit_preceding operation
ANDNOT H340.00  ; 07ST_COMPLETE
AND H340.00  ; 07ST_COMPLETE
ANDNOT H341.00  ; RESISTANCE WORKPIECE
OUT 4405.03  ; Resistance measurement unit_preceding operation
; rung 36
LD 4405.00  ; 07ST_CYCLE RUNNING
IL(002)

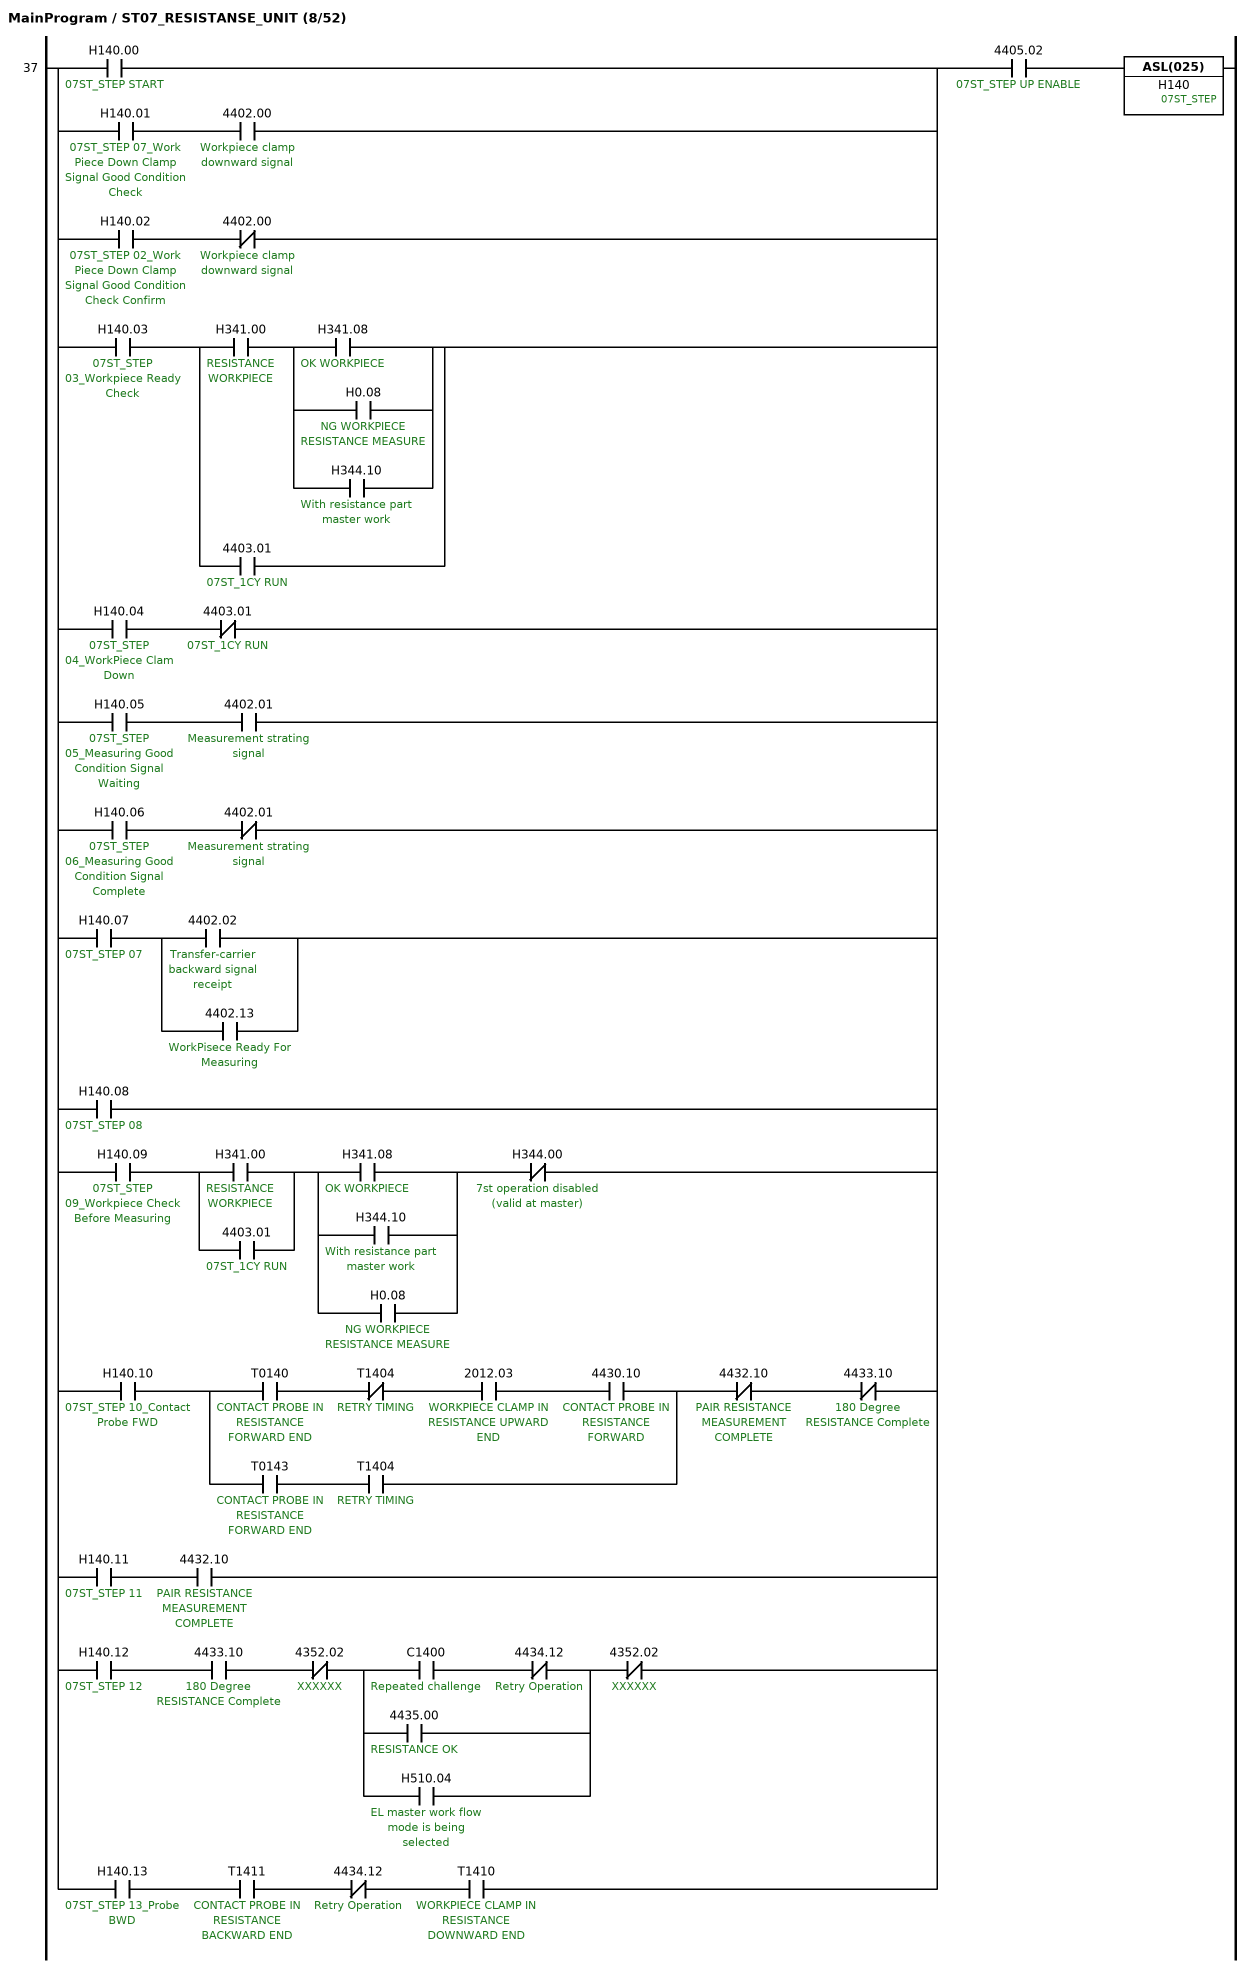
; rung 37
LD H140.00  ; 07ST_STEP START
LD H140.01  ; 07ST_STEP 07_Work Piece Down Clamp Signal Good Condition Check
AND 4402.00  ; Workpiece clamp downward signal
ORLD
LD H140.02  ; 07ST_STEP 02_Work Piece Down Clamp Signal Good Condition Check Confirm
ANDNOT 4402.00  ; Workpiece clamp downward signal
ORLD
LD H140.03  ; 07ST_STEP 03_Workpiece Ready Check
LD H341.00  ; RESISTANCE WORKPIECE
LD H341.08  ; OK WORKPIECE
OR H0.08  ; NG WORKPIECE RESISTANCE MEASURE
OR H344.10  ; With resistance part master work
ANDLD
OR 4403.01  ; 07ST_1CY RUN
ANDLD
ORLD
LD H140.04  ; 07ST_STEP 04_WorkPiece Clam Down
ANDNOT 4403.01  ; 07ST_1CY RUN
ORLD
LD H140.05  ; 07ST_STEP 05_Measuring Good Condition Signal Waiting
AND 4402.01  ; Measurement strating signal
ORLD
LD H140.06  ; 07ST_STEP 06_Measuring Good Condition Signal Complete
ANDNOT 4402.01  ; Measurement strating signal
ORLD
LD H140.07  ; 07ST_STEP 07
LD 4402.02  ; Transfer-carrier backward signal receipt
OR 4402.13  ; WorkPisece Ready For Measuring
ANDLD
ORLD
OR H140.08  ; 07ST_STEP 08
LD H140.09  ; 07ST_STEP 09_Workpiece Check Before Measuring
LD H341.00  ; RESISTANCE WORKPIECE
OR 4403.01  ; 07ST_1CY RUN
ANDLD
LD H341.08  ; OK WORKPIECE
OR H344.10  ; With resistance part master work
OR H0.08  ; NG WORKPIECE RESISTANCE MEASURE
ANDLD
ANDNOT H344.00  ; 7st operation disabled (valid at master)
ORLD
LD H140.10  ; 07ST_STEP 10_Contact Probe FWD
LD T0140  ; CONTACT PROBE IN RESISTANCE FORWARD END
ANDNOT T1404  ; RETRY TIMING
AND 2012.03  ; WORKPIECE CLAMP IN RESISTANCE UPWARD END
AND 4430.10  ; CONTACT PROBE IN RESISTANCE FORWARD
LD T0143  ; CONTACT PROBE IN RESISTANCE FORWARD END
AND T1404  ; RETRY TIMING
ORLD
ANDLD
ANDNOT 4432.10  ; PAIR RESISTANCE MEASUREMENT COMPLETE
ANDNOT 4433.10  ; 180 Degree  RESISTANCE Complete
ORLD
LD H140.11  ; 07ST_STEP 11
AND 4432.10  ; PAIR RESISTANCE MEASUREMENT COMPLETE
ORLD
LD H140.12  ; 07ST_STEP 12
AND 4433.10  ; 180 Degree  RESISTANCE Complete
ANDNOT 4352.02  ; XXXXXX
LD C1400  ; Repeated challenge
ANDNOT 4434.12  ; Retry Operation
OR 4435.00  ; RESISTANCE OK
OR H510.04  ; EL master work flow mode is being selected
ANDLD
ANDNOT 4352.02  ; XXXXXX
ORLD
LD H140.13  ; 07ST_STEP 13_Probe BWD
AND T1411  ; CONTACT PROBE IN RESISTANCE BACKWARD END
ANDNOT 4434.12  ; Retry Operation
AND T1410  ; WORKPIECE CLAMP IN RESISTANCE DOWNWARD END
ORLD
AND 4405.02  ; 07ST_STEP UP ENABLE
ASL(025) H140  ; 07ST_STEP

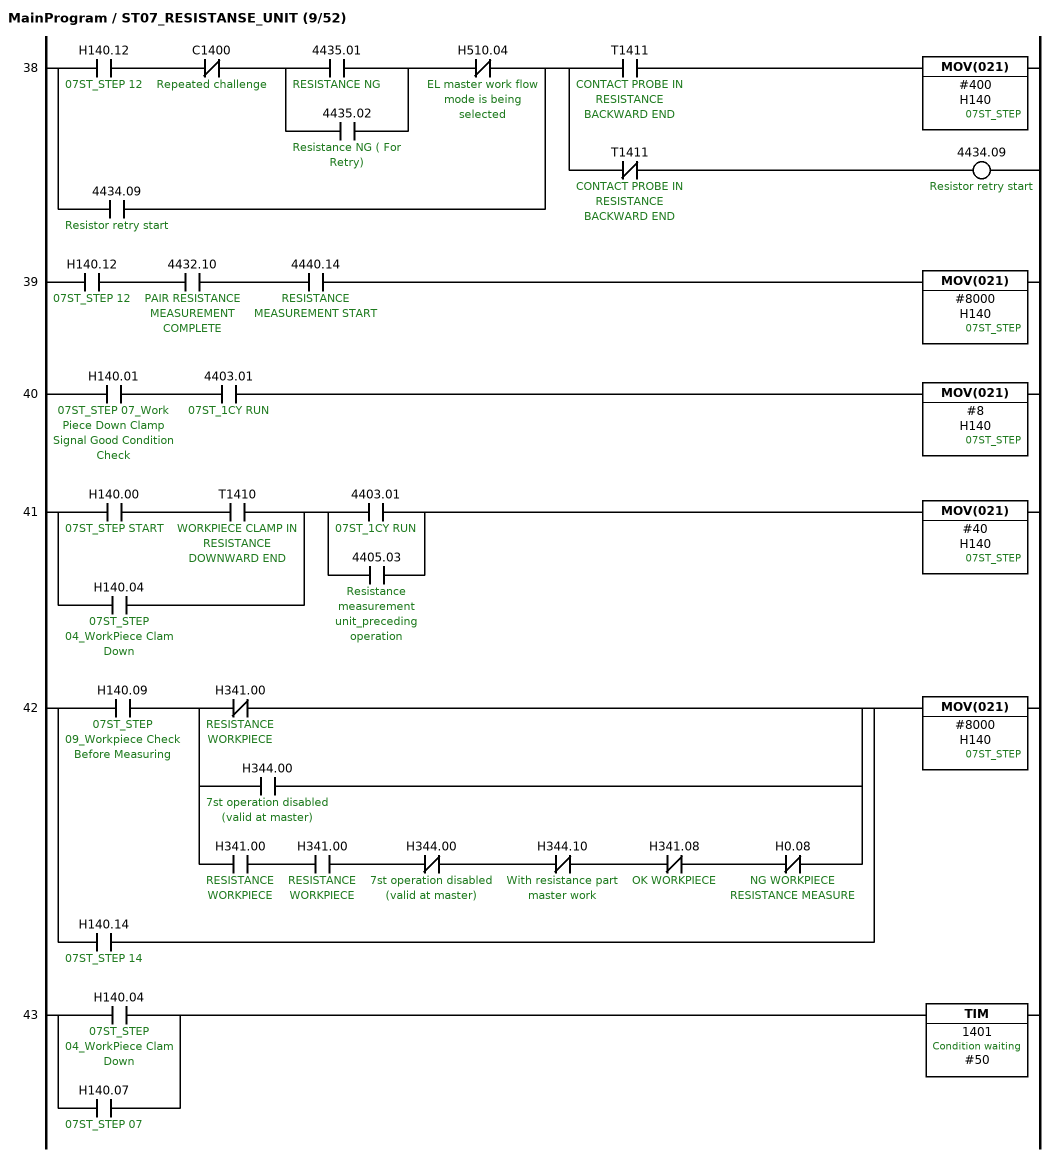
; rung 38
LD H140.12  ; 07ST_STEP 12
ANDNOT C1400  ; Repeated challenge
LD 4435.01  ; RESISTANCE NG
OR 4435.02  ; Resistance NG ( For Retry)
ANDLD
ANDNOT H510.04  ; EL master work flow mode is being selected
OR 4434.09  ; Resistor retry start
OUT TR0
AND T1411  ; CONTACT PROBE IN RESISTANCE BACKWARD END
MOV(021) #400 H140  ; 07ST_STEP
LD TR0
ANDNOT T1411  ; CONTACT PROBE IN RESISTANCE BACKWARD END
OUT 4434.09  ; Resistor retry start
; rung 39
LD H140.12  ; 07ST_STEP 12
AND 4432.10  ; PAIR RESISTANCE MEASUREMENT COMPLETE
AND 4440.14  ; RESISTANCE MEASUREMENT START
MOV(021) #8000 H140  ; 07ST_STEP
; rung 40
LD H140.01  ; 07ST_STEP 07_Work Piece Down Clamp Signal Good Condition Check
AND 4403.01  ; 07ST_1CY RUN
MOV(021) #8 H140  ; 07ST_STEP
; rung 41
LD H140.00  ; 07ST_STEP START
AND T1410  ; WORKPIECE CLAMP IN RESISTANCE DOWNWARD END
OR H140.04  ; 07ST_STEP 04_WorkPiece Clam Down
LD 4403.01  ; 07ST_1CY RUN
OR 4405.03  ; Resistance measurement unit_preceding operation
ANDLD
MOV(021) #40 H140  ; 07ST_STEP
; rung 42
LD H140.09  ; 07ST_STEP 09_Workpiece Check Before Measuring
LDNOT H341.00  ; RESISTANCE WORKPIECE
OR H344.00  ; 7st operation disabled (valid at master)
LD H341.00  ; RESISTANCE WORKPIECE
AND H341.00  ; RESISTANCE WORKPIECE
ANDNOT H344.00  ; 7st operation disabled (valid at master)
ANDNOT H344.10  ; With resistance part master work
ANDNOT H341.08  ; OK WORKPIECE
ANDNOT H0.08  ; NG WORKPIECE RESISTANCE MEASURE
ORLD
ANDLD
OR H140.14  ; 07ST_STEP 14
MOV(021) #8000 H140  ; 07ST_STEP
; rung 43
LD H140.04  ; 07ST_STEP 04_WorkPiece Clam Down
OR H140.07  ; 07ST_STEP 07
TIM 1401 #50  ; Condition waiting

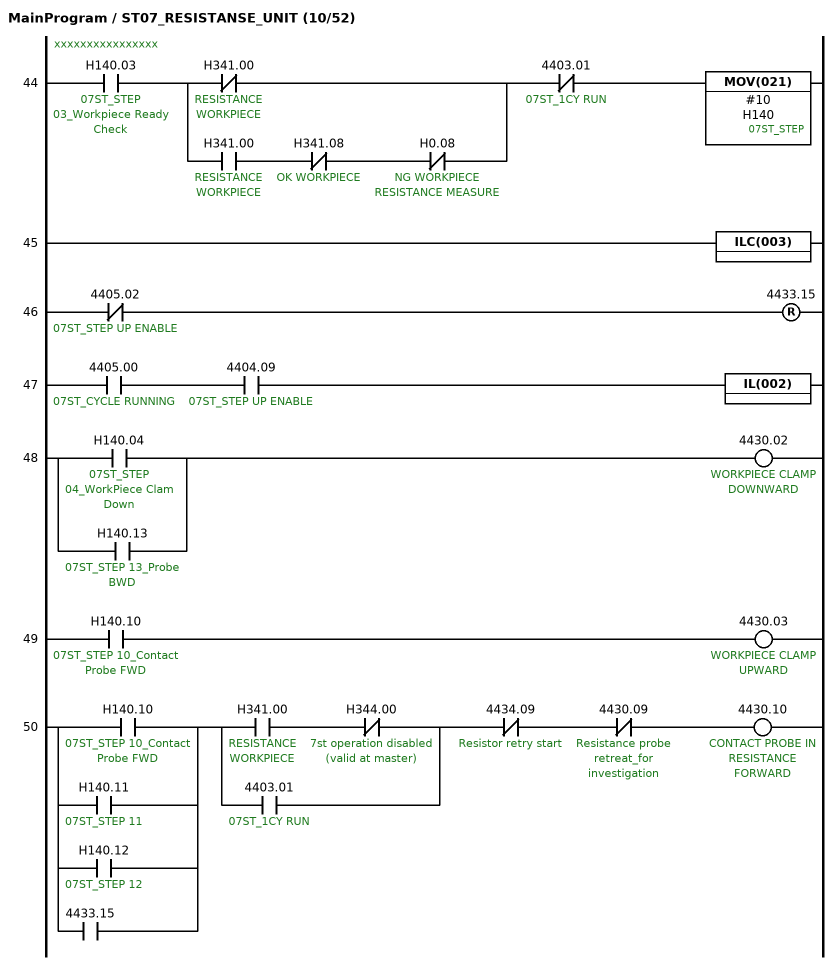
; rung 44: xxxxxxxxxxxxxxxx
LD H140.03  ; 07ST_STEP 03_Workpiece Ready Check
LDNOT H341.00  ; RESISTANCE WORKPIECE
LD H341.00  ; RESISTANCE WORKPIECE
ANDNOT H341.08  ; OK WORKPIECE
ANDNOT H0.08  ; NG WORKPIECE RESISTANCE MEASURE
ORLD
ANDLD
ANDNOT 4403.01  ; 07ST_1CY RUN
MOV(021) #10 H140  ; 07ST_STEP
; rung 45
ILC(003)
; rung 46
LDNOT 4405.02  ; 07ST_STEP UP ENABLE
RSET 4433.15
; rung 47
LD 4405.00  ; 07ST_CYCLE RUNNING
AND 4404.09  ; 07ST_STEP UP ENABLE
IL(002)
; rung 48
LD H140.04  ; 07ST_STEP 04_WorkPiece Clam Down
OR H140.13  ; 07ST_STEP 13_Probe BWD
OUT 4430.02  ; WORKPIECE CLAMP DOWNWARD
; rung 49
LD H140.10  ; 07ST_STEP 10_Contact Probe FWD
OUT 4430.03  ; WORKPIECE CLAMP UPWARD
; rung 50
LD H140.10  ; 07ST_STEP 10_Contact Probe FWD
OR H140.11  ; 07ST_STEP 11
OR H140.12  ; 07ST_STEP 12
OR 4433.15
LD H341.00  ; RESISTANCE WORKPIECE
ANDNOT H344.00  ; 7st operation disabled (valid at master)
OR 4403.01  ; 07ST_1CY RUN
ANDLD
ANDNOT 4434.09  ; Resistor retry start
ANDNOT 4430.09  ; Resistance probe retreat_for investigation
OUT 4430.10  ; CONTACT PROBE IN RESISTANCE FORWARD

